# EPICS substitutions: bpmApp/Db/ai_bpm_pos_erri_cal.substitutions
file ai_bpm_pos_erri_cal.template
{ pattern
	{CN,       N}
	{ "\$(CN)",  "\$(N)" }
}
